PROGRAM Callblocks_FX1_1
VAR
	
FX1_CC1_Clamp_Unit1_3 : clamp;
FX1_CC2_Clamp_Unit2_3 : clamp;
FX1_CC3_Clamp_Unit3_3 : clamp;
FX1_CC4_Clamp_Unit4_3 : clamp;
FX1_CC5_Clamp_Unit5_1 : clamp;
FX1_CC6_Clamp_Unit6_1 : clamp;

Temp_bool : BOOL;
FX1_Feedback_Unit1  : Feedback_FB;
FX1_Feedback_Unit2  : Feedback_FB;
FX1_Feedback_Unit3  : Feedback_FB;
FX1_Feedback_Unit4  : Feedback_FB;
FX1_Feedback_Unit5  : Feedback_FB;
FX1_Feedback_Unit6  : Feedback_FB;


END_VAR
VAR // added by the converter: edge detectors and wires of the graphical bodies
    _w1, _w2, _w3, _w4, _w5, _w6, _w7, _w8 : BOOL;
END_VAR

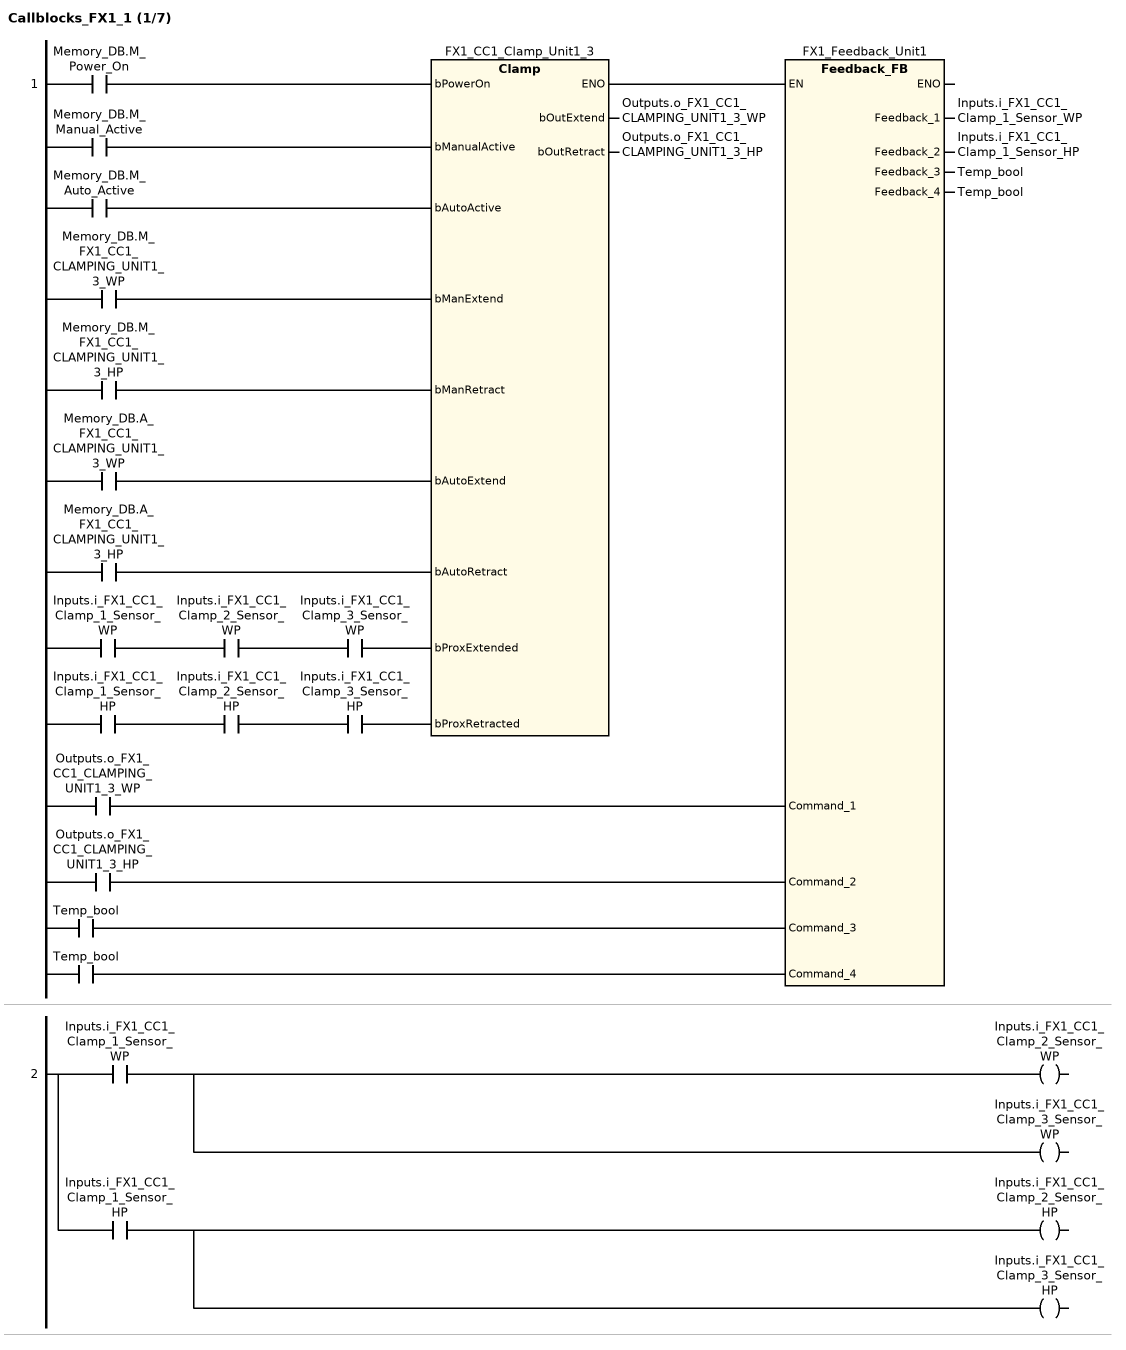
// NETWORK 1
FX1_CC1_Clamp_Unit1_3(
    bPowerOn := Memory_DB.M_Power_On,
    bManualActive := Memory_DB.M_Manual_Active,
    bAutoActive := Memory_DB.M_Auto_Active,
    bManExtend := Memory_DB.M_FX1_CC1_CLAMPING_UNIT1_3_WP,
    bManRetract := Memory_DB.M_FX1_CC1_CLAMPING_UNIT1_3_HP,
    bAutoExtend := Memory_DB.A_FX1_CC1_CLAMPING_UNIT1_3_WP,
    bAutoRetract := Memory_DB.A_FX1_CC1_CLAMPING_UNIT1_3_HP,
    bProxExtended := Inputs.i_FX1_CC1_Clamp_1_Sensor_WP AND Inputs.i_FX1_CC1_Clamp_2_Sensor_WP AND Inputs.i_FX1_CC1_Clamp_3_Sensor_WP,
    bProxRetracted := Inputs.i_FX1_CC1_Clamp_1_Sensor_HP AND Inputs.i_FX1_CC1_Clamp_2_Sensor_HP AND Inputs.i_FX1_CC1_Clamp_3_Sensor_HP,
    bOutExtend => Outputs.o_FX1_CC1_CLAMPING_UNIT1_3_WP,
    bOutRetract => Outputs.o_FX1_CC1_CLAMPING_UNIT1_3_HP); // Clamp
FX1_Feedback_Unit1(
    EN := TRUE,
    Command_1 := Outputs.o_FX1_CC1_CLAMPING_UNIT1_3_WP,
    Command_2 := Outputs.o_FX1_CC1_CLAMPING_UNIT1_3_HP,
    Command_3 := Temp_bool,
    Command_4 := Temp_bool,
    Feedback_1 => Inputs.i_FX1_CC1_Clamp_1_Sensor_WP,
    Feedback_2 => Inputs.i_FX1_CC1_Clamp_1_Sensor_HP,
    Feedback_3 => Temp_bool,
    Feedback_4 => Temp_bool); // Feedback_FB

// NETWORK 2
_w1 := Inputs.i_FX1_CC1_Clamp_1_Sensor_WP;
Inputs.i_FX1_CC1_Clamp_2_Sensor_WP := _w1;
Inputs.i_FX1_CC1_Clamp_3_Sensor_WP := _w1;
_w2 := Inputs.i_FX1_CC1_Clamp_1_Sensor_HP;
Inputs.i_FX1_CC1_Clamp_2_Sensor_HP := _w2;
Inputs.i_FX1_CC1_Clamp_3_Sensor_HP := _w2;

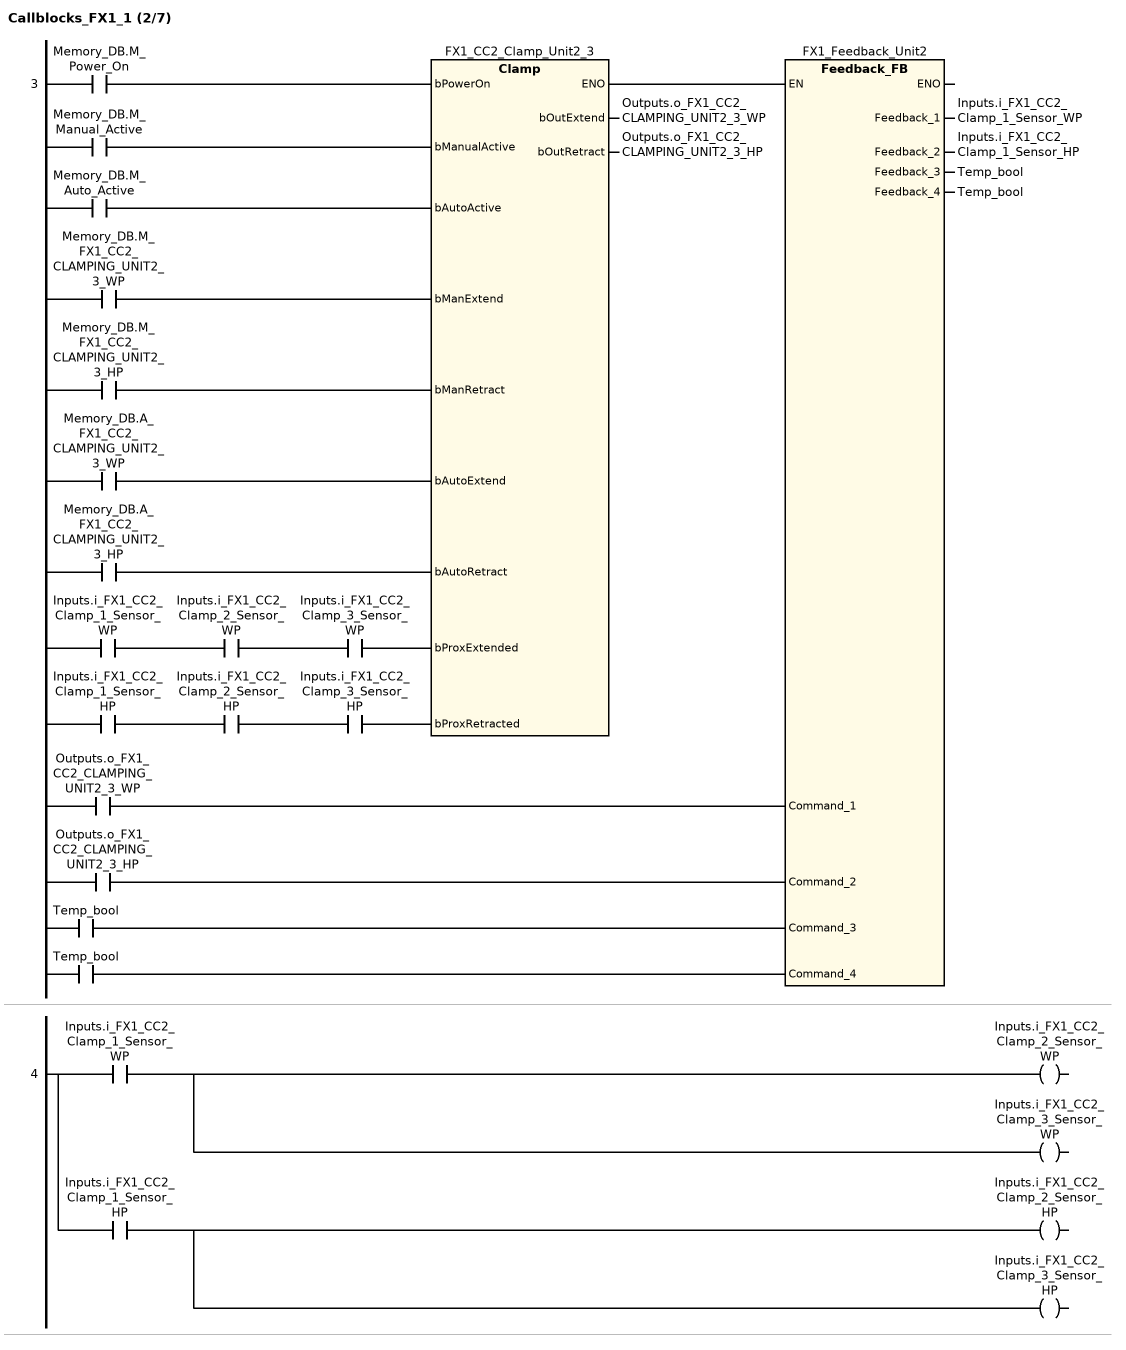
// NETWORK 3
FX1_CC2_Clamp_Unit2_3(
    bPowerOn := Memory_DB.M_Power_On,
    bManualActive := Memory_DB.M_Manual_Active,
    bAutoActive := Memory_DB.M_Auto_Active,
    bManExtend := Memory_DB.M_FX1_CC2_CLAMPING_UNIT2_3_WP,
    bManRetract := Memory_DB.M_FX1_CC2_CLAMPING_UNIT2_3_HP,
    bAutoExtend := Memory_DB.A_FX1_CC2_CLAMPING_UNIT2_3_WP,
    bAutoRetract := Memory_DB.A_FX1_CC2_CLAMPING_UNIT2_3_HP,
    bProxExtended := Inputs.i_FX1_CC2_Clamp_1_Sensor_WP AND Inputs.i_FX1_CC2_Clamp_2_Sensor_WP AND Inputs.i_FX1_CC2_Clamp_3_Sensor_WP,
    bProxRetracted := Inputs.i_FX1_CC2_Clamp_1_Sensor_HP AND Inputs.i_FX1_CC2_Clamp_2_Sensor_HP AND Inputs.i_FX1_CC2_Clamp_3_Sensor_HP,
    bOutExtend => Outputs.o_FX1_CC2_CLAMPING_UNIT2_3_WP,
    bOutRetract => Outputs.o_FX1_CC2_CLAMPING_UNIT2_3_HP); // Clamp
FX1_Feedback_Unit2(
    EN := TRUE,
    Command_1 := Outputs.o_FX1_CC2_CLAMPING_UNIT2_3_WP,
    Command_2 := Outputs.o_FX1_CC2_CLAMPING_UNIT2_3_HP,
    Command_3 := Temp_bool,
    Command_4 := Temp_bool,
    Feedback_1 => Inputs.i_FX1_CC2_Clamp_1_Sensor_WP,
    Feedback_2 => Inputs.i_FX1_CC2_Clamp_1_Sensor_HP,
    Feedback_3 => Temp_bool,
    Feedback_4 => Temp_bool); // Feedback_FB

// NETWORK 4
_w3 := Inputs.i_FX1_CC2_Clamp_1_Sensor_WP;
Inputs.i_FX1_CC2_Clamp_2_Sensor_WP := _w3;
Inputs.i_FX1_CC2_Clamp_3_Sensor_WP := _w3;
_w4 := Inputs.i_FX1_CC2_Clamp_1_Sensor_HP;
Inputs.i_FX1_CC2_Clamp_2_Sensor_HP := _w4;
Inputs.i_FX1_CC2_Clamp_3_Sensor_HP := _w4;

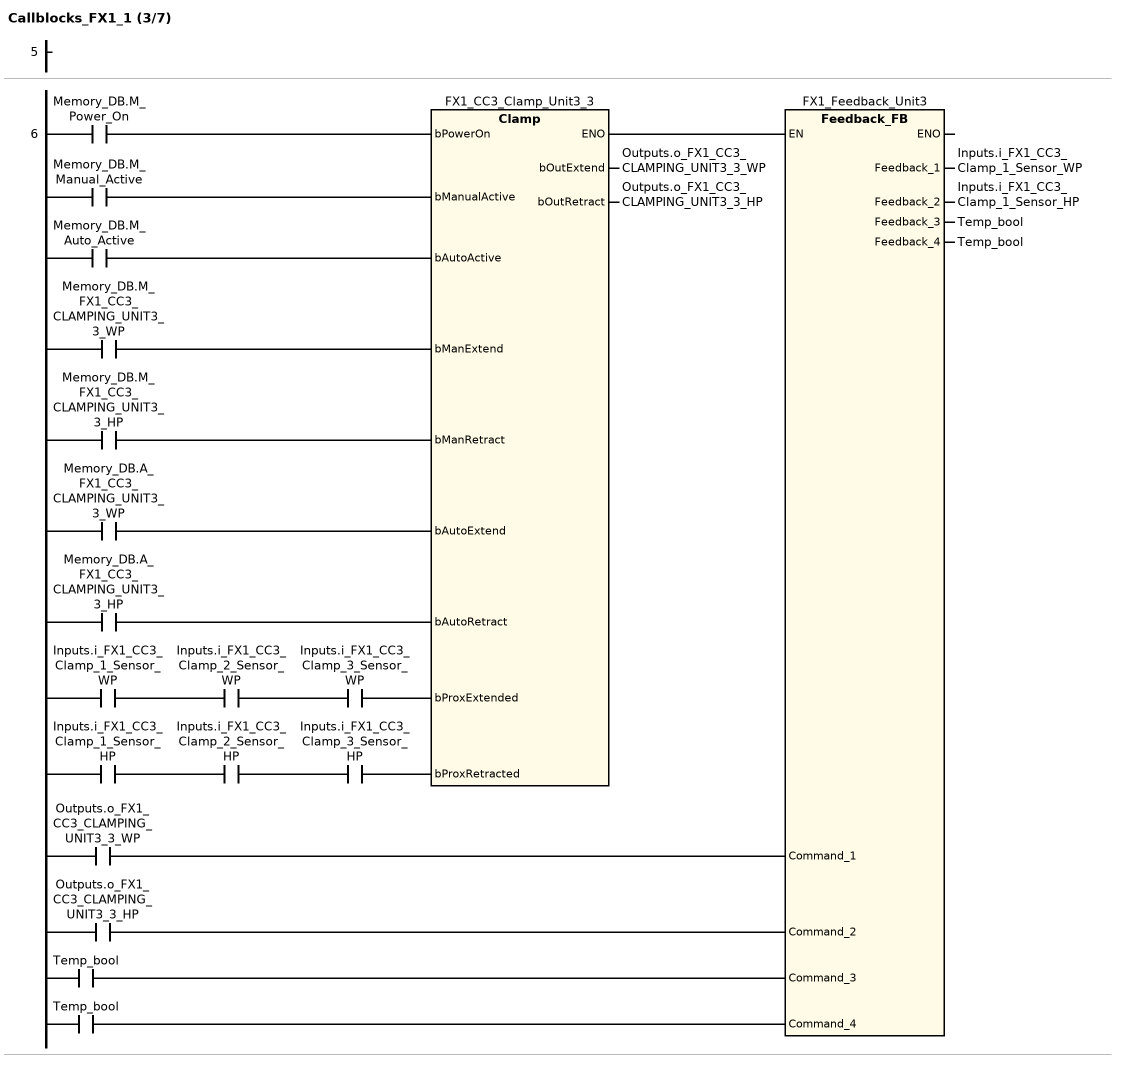
// NETWORK 5

// NETWORK 6
FX1_CC3_Clamp_Unit3_3(
    bPowerOn := Memory_DB.M_Power_On,
    bManualActive := Memory_DB.M_Manual_Active,
    bAutoActive := Memory_DB.M_Auto_Active,
    bManExtend := Memory_DB.M_FX1_CC3_CLAMPING_UNIT3_3_WP,
    bManRetract := Memory_DB.M_FX1_CC3_CLAMPING_UNIT3_3_HP,
    bAutoExtend := Memory_DB.A_FX1_CC3_CLAMPING_UNIT3_3_WP,
    bAutoRetract := Memory_DB.A_FX1_CC3_CLAMPING_UNIT3_3_HP,
    bProxExtended := Inputs.i_FX1_CC3_Clamp_1_Sensor_WP AND Inputs.i_FX1_CC3_Clamp_2_Sensor_WP AND Inputs.i_FX1_CC3_Clamp_3_Sensor_WP,
    bProxRetracted := Inputs.i_FX1_CC3_Clamp_1_Sensor_HP AND Inputs.i_FX1_CC3_Clamp_2_Sensor_HP AND Inputs.i_FX1_CC3_Clamp_3_Sensor_HP,
    bOutExtend => Outputs.o_FX1_CC3_CLAMPING_UNIT3_3_WP,
    bOutRetract => Outputs.o_FX1_CC3_CLAMPING_UNIT3_3_HP); // Clamp
FX1_Feedback_Unit3(
    EN := TRUE,
    Command_1 := Outputs.o_FX1_CC3_CLAMPING_UNIT3_3_WP,
    Command_2 := Outputs.o_FX1_CC3_CLAMPING_UNIT3_3_HP,
    Command_3 := Temp_bool,
    Command_4 := Temp_bool,
    Feedback_1 => Inputs.i_FX1_CC3_Clamp_1_Sensor_WP,
    Feedback_2 => Inputs.i_FX1_CC3_Clamp_1_Sensor_HP,
    Feedback_3 => Temp_bool,
    Feedback_4 => Temp_bool); // Feedback_FB

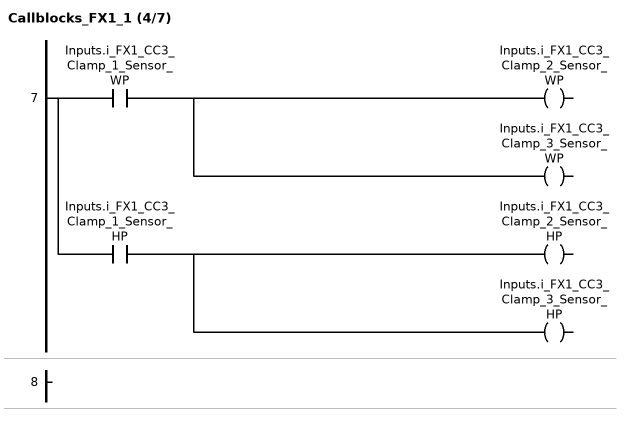
// NETWORK 7
_w5 := Inputs.i_FX1_CC3_Clamp_1_Sensor_WP;
Inputs.i_FX1_CC3_Clamp_2_Sensor_WP := _w5;
Inputs.i_FX1_CC3_Clamp_3_Sensor_WP := _w5;
_w6 := Inputs.i_FX1_CC3_Clamp_1_Sensor_HP;
Inputs.i_FX1_CC3_Clamp_2_Sensor_HP := _w6;
Inputs.i_FX1_CC3_Clamp_3_Sensor_HP := _w6;

// NETWORK 8

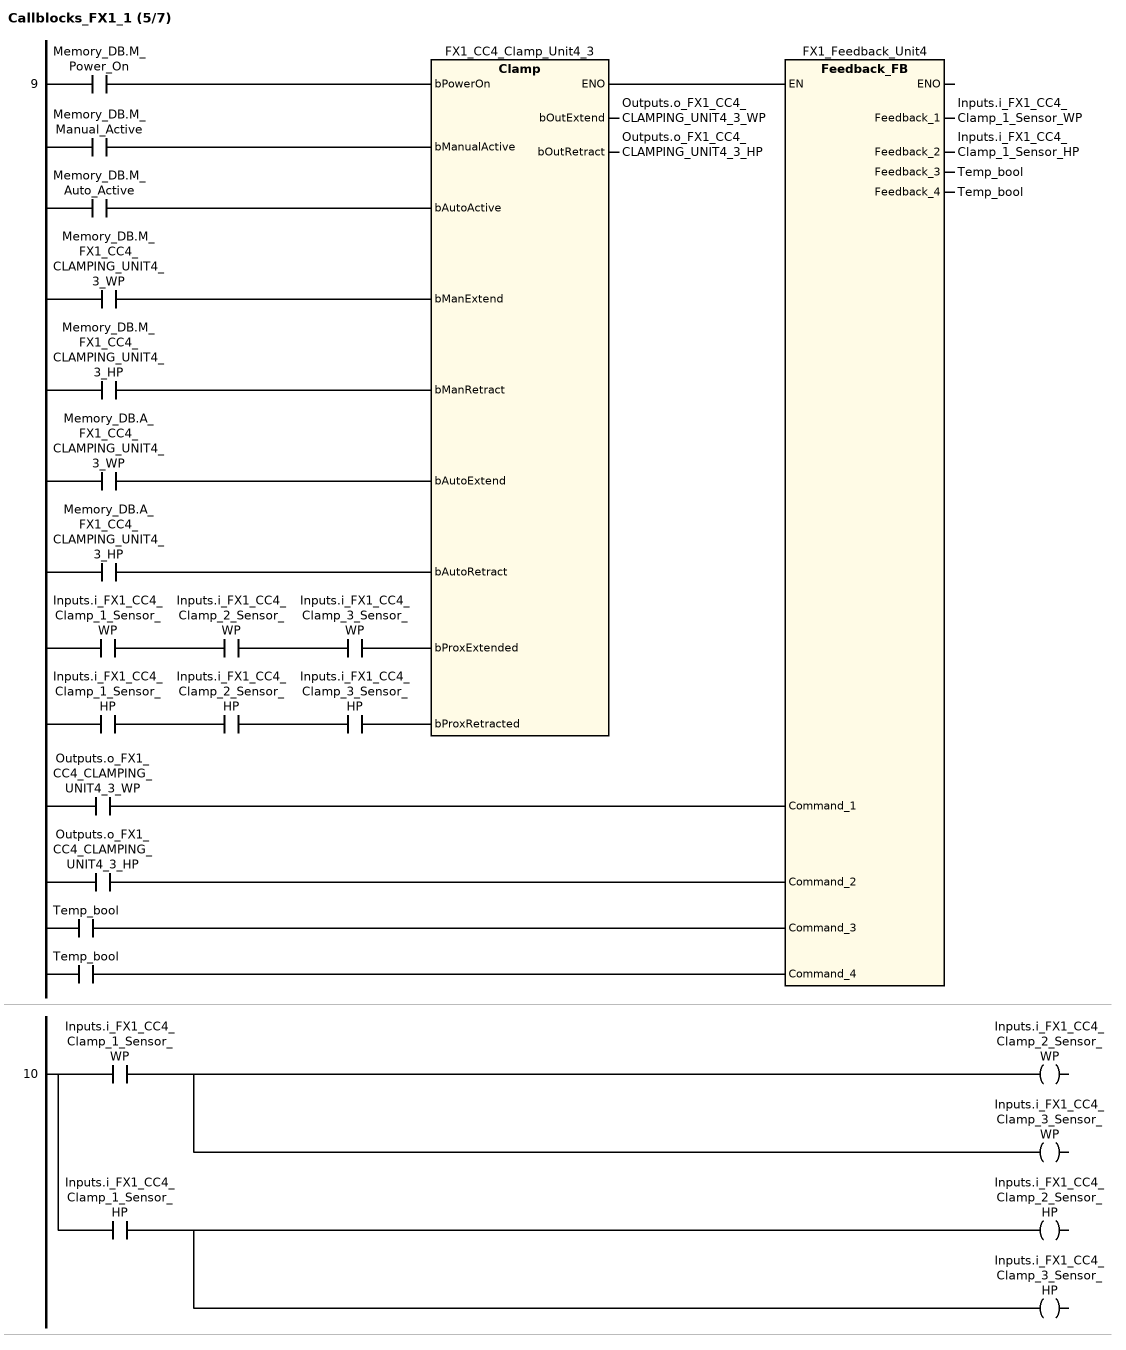
// NETWORK 9
FX1_CC4_Clamp_Unit4_3(
    bPowerOn := Memory_DB.M_Power_On,
    bManualActive := Memory_DB.M_Manual_Active,
    bAutoActive := Memory_DB.M_Auto_Active,
    bManExtend := Memory_DB.M_FX1_CC4_CLAMPING_UNIT4_3_WP,
    bManRetract := Memory_DB.M_FX1_CC4_CLAMPING_UNIT4_3_HP,
    bAutoExtend := Memory_DB.A_FX1_CC4_CLAMPING_UNIT4_3_WP,
    bAutoRetract := Memory_DB.A_FX1_CC4_CLAMPING_UNIT4_3_HP,
    bProxExtended := Inputs.i_FX1_CC4_Clamp_1_Sensor_WP AND Inputs.i_FX1_CC4_Clamp_2_Sensor_WP AND Inputs.i_FX1_CC4_Clamp_3_Sensor_WP,
    bProxRetracted := Inputs.i_FX1_CC4_Clamp_1_Sensor_HP AND Inputs.i_FX1_CC4_Clamp_2_Sensor_HP AND Inputs.i_FX1_CC4_Clamp_3_Sensor_HP,
    bOutExtend => Outputs.o_FX1_CC4_CLAMPING_UNIT4_3_WP,
    bOutRetract => Outputs.o_FX1_CC4_CLAMPING_UNIT4_3_HP); // Clamp
FX1_Feedback_Unit4(
    EN := TRUE,
    Command_1 := Outputs.o_FX1_CC4_CLAMPING_UNIT4_3_WP,
    Command_2 := Outputs.o_FX1_CC4_CLAMPING_UNIT4_3_HP,
    Command_3 := Temp_bool,
    Command_4 := Temp_bool,
    Feedback_1 => Inputs.i_FX1_CC4_Clamp_1_Sensor_WP,
    Feedback_2 => Inputs.i_FX1_CC4_Clamp_1_Sensor_HP,
    Feedback_3 => Temp_bool,
    Feedback_4 => Temp_bool); // Feedback_FB

// NETWORK 10
_w7 := Inputs.i_FX1_CC4_Clamp_1_Sensor_WP;
Inputs.i_FX1_CC4_Clamp_2_Sensor_WP := _w7;
Inputs.i_FX1_CC4_Clamp_3_Sensor_WP := _w7;
_w8 := Inputs.i_FX1_CC4_Clamp_1_Sensor_HP;
Inputs.i_FX1_CC4_Clamp_2_Sensor_HP := _w8;
Inputs.i_FX1_CC4_Clamp_3_Sensor_HP := _w8;

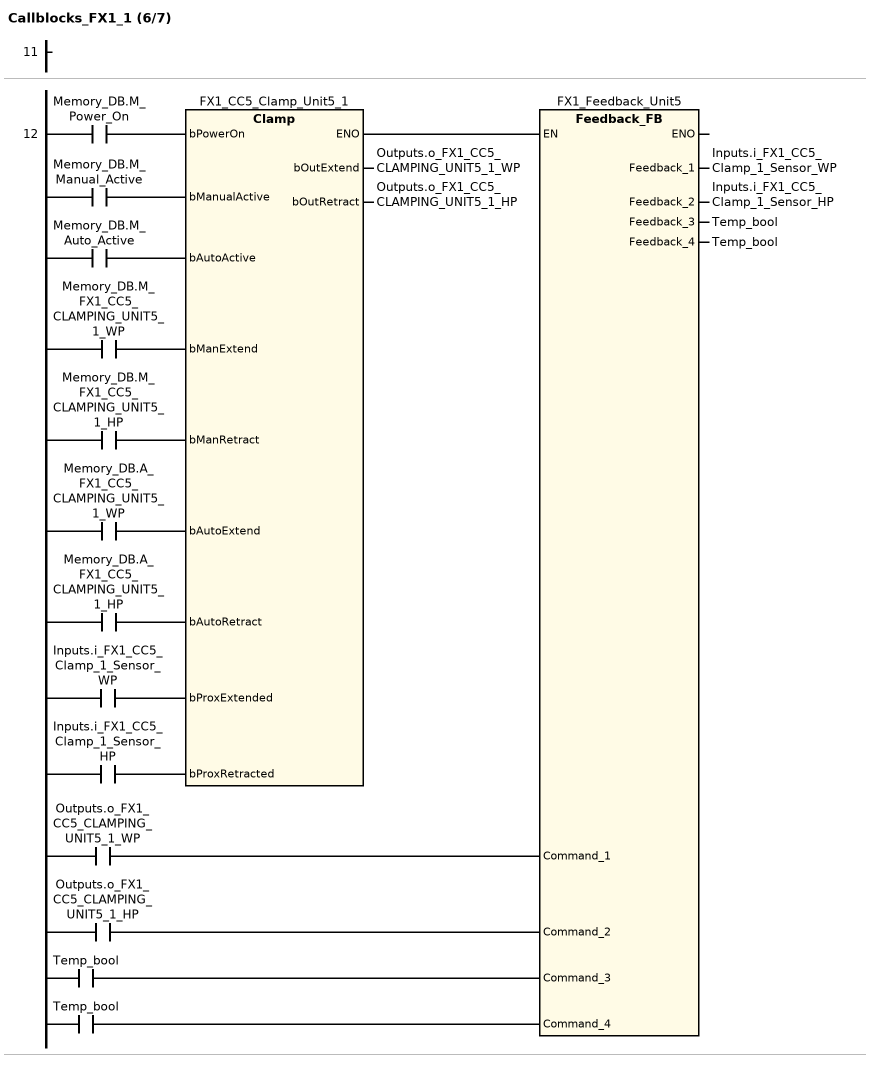
// NETWORK 11

// NETWORK 12
FX1_CC5_Clamp_Unit5_1(
    bPowerOn := Memory_DB.M_Power_On,
    bManualActive := Memory_DB.M_Manual_Active,
    bAutoActive := Memory_DB.M_Auto_Active,
    bManExtend := Memory_DB.M_FX1_CC5_CLAMPING_UNIT5_1_WP,
    bManRetract := Memory_DB.M_FX1_CC5_CLAMPING_UNIT5_1_HP,
    bAutoExtend := Memory_DB.A_FX1_CC5_CLAMPING_UNIT5_1_WP,
    bAutoRetract := Memory_DB.A_FX1_CC5_CLAMPING_UNIT5_1_HP,
    bProxExtended := Inputs.i_FX1_CC5_Clamp_1_Sensor_WP,
    bProxRetracted := Inputs.i_FX1_CC5_Clamp_1_Sensor_HP,
    bOutExtend => Outputs.o_FX1_CC5_CLAMPING_UNIT5_1_WP,
    bOutRetract => Outputs.o_FX1_CC5_CLAMPING_UNIT5_1_HP); // Clamp
FX1_Feedback_Unit5(
    EN := TRUE,
    Command_1 := Outputs.o_FX1_CC5_CLAMPING_UNIT5_1_WP,
    Command_2 := Outputs.o_FX1_CC5_CLAMPING_UNIT5_1_HP,
    Command_3 := Temp_bool,
    Command_4 := Temp_bool,
    Feedback_1 => Inputs.i_FX1_CC5_Clamp_1_Sensor_WP,
    Feedback_2 => Inputs.i_FX1_CC5_Clamp_1_Sensor_HP,
    Feedback_3 => Temp_bool,
    Feedback_4 => Temp_bool); // Feedback_FB

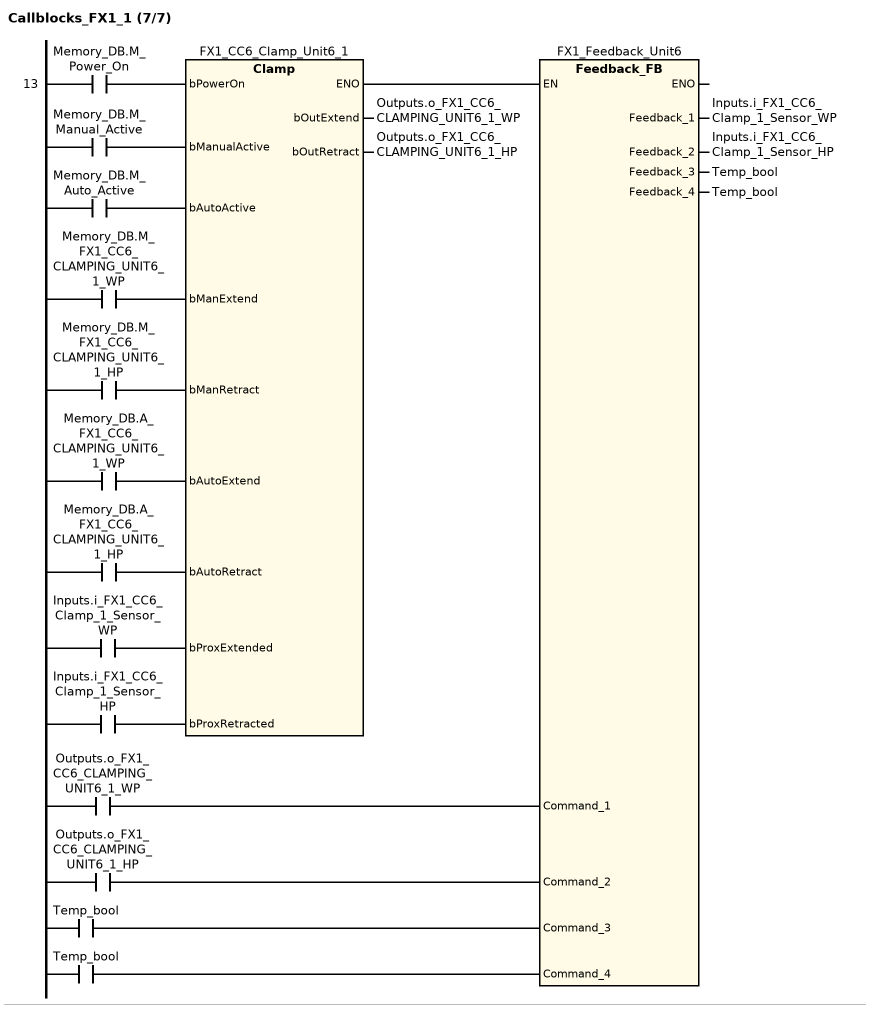
// NETWORK 13
FX1_CC6_Clamp_Unit6_1(
    bPowerOn := Memory_DB.M_Power_On,
    bManualActive := Memory_DB.M_Manual_Active,
    bAutoActive := Memory_DB.M_Auto_Active,
    bManExtend := Memory_DB.M_FX1_CC6_CLAMPING_UNIT6_1_WP,
    bManRetract := Memory_DB.M_FX1_CC6_CLAMPING_UNIT6_1_HP,
    bAutoExtend := Memory_DB.A_FX1_CC6_CLAMPING_UNIT6_1_WP,
    bAutoRetract := Memory_DB.A_FX1_CC6_CLAMPING_UNIT6_1_HP,
    bProxExtended := Inputs.i_FX1_CC6_Clamp_1_Sensor_WP,
    bProxRetracted := Inputs.i_FX1_CC6_Clamp_1_Sensor_HP,
    bOutExtend => Outputs.o_FX1_CC6_CLAMPING_UNIT6_1_WP,
    bOutRetract => Outputs.o_FX1_CC6_CLAMPING_UNIT6_1_HP); // Clamp
FX1_Feedback_Unit6(
    EN := TRUE,
    Command_1 := Outputs.o_FX1_CC6_CLAMPING_UNIT6_1_WP,
    Command_2 := Outputs.o_FX1_CC6_CLAMPING_UNIT6_1_HP,
    Command_3 := Temp_bool,
    Command_4 := Temp_bool,
    Feedback_1 => Inputs.i_FX1_CC6_Clamp_1_Sensor_WP,
    Feedback_2 => Inputs.i_FX1_CC6_Clamp_1_Sensor_HP,
    Feedback_3 => Temp_bool,
    Feedback_4 => Temp_bool); // Feedback_FB

END_PROGRAM

(* stored: Version 1.1.0.1, ProductVersion 3.1.4024.16
   POU Callblocks_FX1_1: Id {846d5464-2330-4a13-bbc5-7afed2a9ce36}, SpecialFunc None *)
